TYPE E_SecondaryCriterionAction : (
    SECONDARY_ADVANCE_AND_NOK := 0,
    SECONDARY_CONTROLLED_EXIT_NOK := 10
); END_TYPE

(* stored: Version 1.1.0.1
   DUT E_SecondaryCriterionAction: Id {E3000000-0000-4000-8000-000000000011} *)
